PROGRAM PID_Difference_ctrl
VAR
		lrDiff: LREAL;
	lrPrevious: LREAL;
	lrOutput: LREAL;
END_VAR

lrDiff := PID_ctrl.rPump3_Freq_Reading_Raw - lrPrevious;
lrPrevious := PID_ctrl.rPump3_Freq_Reading_Raw ;

IF	lrOutput + lrDiff > 0 AND  lrOutput + lrDiff < 32767 THEN
	lrOutput := lrOutput + lrDiff;
ELSIF lrDiff > 0 THEN
	lrOutput := 32767;	
	
ELSIF lrDiff < 0 THEN
	lrOutput := 0;	
	
END_IF

PID_ctrl.Stn3FlowRawData;
PID_ctrl.Stn3ActualFlowRawData;

END_PROGRAM

(* stored: Version 1.1.0.1, ProductVersion 3.1.4024.12
   POU PID_Difference_ctrl: Id {22fdeb07-2eee-48c5-8035-c5216089ad1d}, SpecialFunc None *)
